// TIA Portal V20 export
// export: Created 2025-12-01T14:57:44.7906699Z, ExportSetting None, DisplayName Totally Integrated Automation Portal, DisplayVersion V20 Update 3, DisplayName TIA Portal Openness, DisplayVersion V20 Update 3, DisplayName TIA Portal Version Control Interface, DisplayVersion V20 Update 3, DisplayName STEP 7 Professional, DisplayVersion V20 Update 3, DisplayName STEP 7 Safety, DisplayVersion V20 Update 2, DisplayName WinCC Basic/Comfort/Advanced, DisplayVersion V20 Update 3, DisplayName WinCC Professional, DisplayVersion V20 Update 3, DisplayName WinCC Unified, DisplayVersion V20 Update 3
FUNCTION "FC716_Router_BuscarEtiqueta_Lint_y_sacar_orden" : Void   // FC716, SCL
{ S7_Optimized_Access := 'FALSE' }
// stored: AutoNumber false, SetENOAutomatically false
   VAR_INPUT
      Etiqueta : ULInt;   // Etiqueta A Buscar en la Base de Datos
      Numero_SCR : UInt;
   END_VAR
   VAR_TEMP
      Cola : UDInt;
      EtiquetaTMP : ULInt;
      Posicion_Etiqueta_TMP : UInt;
      aux_pos : UInt;
      Num_Inic : UInt;
      Tipo_SCR : UInt;
      primer_bit : UInt;
      numero_bits : UInt;
      contador : UInt;
      CERO : Byte;
      Retval : Int;
      orden : Byte;
      orden_aux AT orden : Array[0..7] of Bool;
      cont_aux : UInt;
      Inic_bits : Array[1..8] of Bool;
      Reg_Etiq_Temp : "ROUT_Reg_Etiqueta";
      Datos_fifo : "ROUT_Orden_Fifo_Scanner";
      datos_actuales_fifo : "ROUT_Orden_Fifo_Scanner";
   END_VAR
BEGIN
   REGION inicilizar

       #EtiquetaTMP := #Etiqueta;
       #Posicion_Etiqueta_TMP := 0;
       #CERO := 0;
       #Num_Inic := "DB912_Tipo_Scanner_Router".SCANNER[#Numero_SCR].Num_Inicializacion;
       #Tipo_SCR := "DB912_Tipo_Scanner_Router".SCANNER[#Numero_SCR].Tipo;
       #Retval:=FILL(BVAL := #CERO, BLK => #Datos_fifo);
       SCATTER(IN := "Estado_inicializacion",
               OUT => #Inic_bits);


   END_REGION
   REGION comprobar_inicializacion
       // comprobamos si el scanner que estamos comprobando está en proceso de inicialización
       IF ((#Num_Inic >= 1) AND (#Num_Inic <= 8)) THEN
           // si tiene un numero de inicialización configurado, comprobamos si está activo
           IF (#Inic_bits[#Num_Inic] = true) THEN
               GOTO proceso_INIC;
           END_IF;
       END_IF;

   END_REGION

   REGION comprobar_etiqueta

       IF #EtiquetaTMP <= 0 THEN
           GOTO error_lectura;
       ELSE
           #Cola := #EtiquetaTMP MOD "ROUT_N_Colas";        // calculamos el numero de cola
       END_IF;
   END_REGION

   #Posicion_Etiqueta_TMP := "DB212_Cola_Activa".Cola[#Cola];

   // comprobamos si existe alguna etiqueta en esa cola

   elegir_db_busqueda:

       // si esa etiqueta no está dada de alta en las colas es que no está activa 
   IF #Posicion_Etiqueta_TMP = 0 THEN
       GOTO lectura_NENC;
   END_IF;


   REGION elegir_db_busqueda
       CASE #Posicion_Etiqueta_TMP OF
           1..1000:
               GOTO busca_1_999;
           1001..2000:
               GOTO busca_1k;
           2001..3000:
               GOTO busca_2k;
           3001..4000:
               GOTO busca_3k;
           ELSE

               GOTO lectura_NENC;
       END_CASE;
   END_REGION

   ////////////////////////////////////////////
   REGION busca_1_a_1000
   busca_1_999:
       IF #EtiquetaTMP = "DB201_RegEtiquetas_0001_1000".Reg_Etiqueta[#Posicion_Etiqueta_TMP].CDB THEN
           #Reg_Etiq_Temp := "DB201_RegEtiquetas_0001_1000".Reg_Etiqueta[#Posicion_Etiqueta_TMP];
           GOTO lectura_encontrada;
       ELSE
           #Posicion_Etiqueta_TMP := "DB201_RegEtiquetas_0001_1000".Reg_Etiqueta[#Posicion_Etiqueta_TMP].Posterior;
           GOTO elegir_db_busqueda;
       END_IF;
   END_REGION

   ////////////////////////////////////////////
   REGION busca_1001_a_2000
   busca_1k:
       #Posicion_Etiqueta_TMP := #Posicion_Etiqueta_TMP - 1000;
       IF #EtiquetaTMP = "DB202_RegEtiquetas_1001_2000".Reg_Etiqueta[#Posicion_Etiqueta_TMP].CDB THEN
           #Reg_Etiq_Temp := "DB202_RegEtiquetas_1001_2000".Reg_Etiqueta[#Posicion_Etiqueta_TMP];
           GOTO lectura_encontrada;
       ELSE
           #Posicion_Etiqueta_TMP := "DB202_RegEtiquetas_1001_2000".Reg_Etiqueta[#Posicion_Etiqueta_TMP].Posterior;
           GOTO elegir_db_busqueda;
       END_IF;
   END_REGION

   ////////////////////////////////////////////
   REGION busca_2001_a_3000
   busca_2k:
       #Posicion_Etiqueta_TMP := #Posicion_Etiqueta_TMP - 2000;
       IF #EtiquetaTMP = "DB203_RegEtiquetas_2001_3000".Reg_Etiqueta[#Posicion_Etiqueta_TMP].CDB THEN
           #Reg_Etiq_Temp := "DB203_RegEtiquetas_2001_3000".Reg_Etiqueta[#Posicion_Etiqueta_TMP];
           GOTO lectura_encontrada;
       ELSE
           #Posicion_Etiqueta_TMP := "DB203_RegEtiquetas_2001_3000".Reg_Etiqueta[#Posicion_Etiqueta_TMP].Posterior;
           GOTO elegir_db_busqueda;
       END_IF;

   END_REGION

   ////////////////////////////////////////////
   REGION busca_3001_a_4000
   busca_3k:
       #Posicion_Etiqueta_TMP := #Posicion_Etiqueta_TMP - 3000;
       IF #EtiquetaTMP = "DB204_RegEtiquetas_3001_4000".Reg_Etiqueta[#Posicion_Etiqueta_TMP].CDB THEN
           #Reg_Etiq_Temp := "DB204_RegEtiquetas_3001_4000".Reg_Etiqueta[#Posicion_Etiqueta_TMP];
           GOTO lectura_encontrada;
       ELSE
           #Posicion_Etiqueta_TMP := "DB204_RegEtiquetas_3001_4000".Reg_Etiqueta[#Posicion_Etiqueta_TMP].Posterior;
           GOTO elegir_db_busqueda;
       END_IF
       ;
   END_REGION

   REGION Especial_error_lectura
   error_lectura:
       #Reg_Etiq_Temp := "DB209_Reg_Etquetas_Esp_Activa".Reg_Etiqueta[1];
       #Datos_fifo.Orden := w#16#90;
       IF #Tipo_SCR = 2 THEN // tipo validación
           #Datos_fifo.Identificador := #Etiqueta;
           GOTO guardar_orden;
       END_IF;
       GOTO extraer_orden;
   END_REGION
   REGION Especial_NENC
   lectura_NENC:
       #Datos_fifo.Identificador := #Etiqueta;
       IF (#Tipo_SCR = 2) THEN
           #Datos_fifo.Orden := w#16#80;

           GOTO guardar_orden;
       END_IF;
       #Reg_Etiq_Temp := "DB209_Reg_Etquetas_Esp_Activa".Reg_Etiqueta[2];
       #Datos_fifo.Orden := w#16#A0;
       // hay dos casos posibles. si el escanner es normal extrae orden normal
       // si es de validacion de etiqueta, extrae el predeterminado
       GOTO extraer_orden;
   END_REGION
   REGION Especial_INIC
   proceso_INIC:
       #Reg_Etiq_Temp := "DB209_Reg_Etquetas_Esp_Activa".Reg_Etiqueta[3];
       #Datos_fifo.Orden := w#16#C0;
       GOTO extraer_orden;
   END_REGION
   REGION lectura_ok
   lectura_encontrada:
       #Datos_fifo.Identificador := #Etiqueta;
       IF #Tipo_SCR = 2 THEN
           #Datos_fifo.Orden := w#16#81;
           GOTO guardar_orden;
       ELSE
           #Datos_fifo.Orden := w#16#80;
           GOTO extraer_orden;
       END_IF;


   END_REGION

   REGION Extraer orden
   extraer_orden:
       #Datos_fifo.Identificador := #Etiqueta;
   // proceso extracción de la orden
   // miramos cual es el primer bit que tenemos que sacar de la orden
       #primer_bit := "DB912_Tipo_Scanner_Router".SCANNER[#Numero_SCR].Bit_Ini_Ordenes;
       #numero_bits := "DB912_Tipo_Scanner_Router".SCANNER[#Numero_SCR].N_Bits_Orden;
       #cont_aux := 0;
       #orden := #Datos_fifo.Orden;
       FOR #contador := #primer_bit TO (#primer_bit + #numero_bits - 1) DO
           #orden_aux[#cont_aux] := #Reg_Etiq_Temp.BIT_Orden[#contador];
           #cont_aux += 1;
       END_FOR;
       #Datos_fifo.Orden := #orden;
       ;
   END_REGION

   REGION Guardar_Orden
   guardar_orden:
       // miramos si ya hay algo en la fifo
       "FC571_Leer_Datos_Fifo"(DB_FIFO_Ordenes:="ROUT_NDB_FIFO_Odr_SCR",
                               Num_Scanner:=#Numero_SCR,
                               Long_FIFO:=1,
                               Posicion_FIFO:=1,
                               Datos_Scanner_Cruce=>#datos_actuales_fifo);

       IF #datos_actuales_fifo.Orden <> 0 THEN
           #Datos_fifo.Orden := w#16#FF;
       END_IF;
       "FC572_Guardar_Datos_Fifo"(DB_FIFO_Ordenes:="ROUT_NDB_FIFO_Odr_SCR",
                                  Num_Scanner:=#Numero_SCR,
                                  Long_FIFO:=1,
                                  Posicion_FIFO:=1,
                                  Datos_Scanner_Cruce:=#Datos_fifo);

       // lo ultimo es borrar la N de la nueva lectura en el db211   ;
       // 
       "DB211_Lecturas_Scanner".Lec_Scanner[#Numero_SCR].Lectura_SCR[0]:= l#0;



   END_REGION
END_FUNCTION
